// TIA Portal V14 SP1 export
// export: Created 2017-11-15T10:09:22.8590153Z, ExportSetting WithDefaults, DisplayName Totally Integrated Automation Portal, DisplayVersion V14 SP1 Update 3, DisplayName TIA Portal Openness, DisplayVersion V14 SP1 Update 2, DisplayName STEP 7 Professional, DisplayVersion V14 SP1 Update 3, DisplayName SIMATIC Energy Suite, DisplayVersion V14 SP1 Update 2, DisplayName WinCC Professional, DisplayVersion V14 SP1 Update 3
VAR_GLOBAL   // PLC tag table "MyTagTable"
   Moto_DI0 AT %I0.0 : Bool;   // 0号电机准备好
   Moto_DI1 AT %I0.1 : Bool;   // 1号电机准备好
   Moto_DI2 AT %I0.2 : Bool;   // 2号电机准备好
   Moto_DI3 AT %I0.3 : Bool;   // 3号电机准备好
   Moto_DI4 AT %I0.4 : Bool;   // 4号电机准备好
   Moto_DI5 AT %I0.5 : Bool;   // 5号电机准备好
   Moto_DI6 AT %I0.6 : Bool;   // 6号电机准备好
   Moto_DI7 AT %I0.7 : Bool;   // 7号电机准备好
   Moto_DO0 AT %Q0.0 : Bool;   // 0号电机开启
   Moto_DO1 AT %Q0.1 : Bool;   // 1号电机开启
   Moto_DO2 AT %Q0.2 : Bool;   // 2号电机开启
   Moto_DO3 AT %Q0.3 : Bool;   // 3号电机开启
   Moto_DO4 AT %Q0.4 : Bool;   // 4号电机开启
   Moto_DO5 AT %Q0.5 : Bool;   // 5号电机开启
   Moto_DO6 AT %Q0.6 : Bool;   // 6号电机开启
   Moto_DO7 AT %Q0.7 : Bool;   // 7号电机开启
   Moto_AI0 AT %IW2 : Int;   // 0号电机速度反馈
   Moto_AI1 AT %IW4 : Int;   // 1号电机速度反馈
   Moto_AI2 AT %IW6 : Int;   // 2号电机速度反馈
   Moto_AI3 AT %IW8 : Int;   // 3号电机速度反馈
   Moto_AI4 AT %IW10 : Int;   // 4号电机速度反馈
   Moto_AI5 AT %IW12 : Int;   // 5号电机速度反馈
   Moto_AI6 AT %IW14 : Int;   // 6号电机速度反馈
   Moto_AI7 AT %IW16 : Int;   // 7号电机速度反馈
   Moto_AO0 AT %QW1 : Int;   // 0号电机速度给定
   Moto_AO1 AT %QW3 : Int;   // 1号电机速度给定
   Moto_AO2 AT %QW5 : Int;   // 2号电机速度给定
   Moto_AO3 AT %QW7 : Int;   // 3号电机速度给定
END_VAR
